{attribute 'linkalways'} 
{attribute 'no_explicit_call' := 'This FB is a CLASS and must be accessed using methods or properties'}
{attribute 'enable_dynamic_creation'}
FUNCTION_BLOCK _ETcVnFontType EXTENDS EnumDatatypeBase
VAR
	localData : ETcVnFontType;
	activeData : REFERENCE TO ETcVnFontType;
	enumBaseDatatype : _DINT(localData);
END_VAR

METHOD PRIVATE AddLocalEnumeration
VAR_INPUT
	Enumeration : T_MAXSTRING;
	Value : ETcVnFontType;
END_VAR
AddEnumeration(Enumeration, Value);
END_METHOD

PROPERTY PUBLIC Address : PVOID
GET
Address := ADR(activeData);
END_GET
END_PROPERTY

METHOD PUBLIC ClearReference
VAR_INPUT
END_VAR
activeData REF= localData;
SetBaseDatatypeReference();
END_METHOD

METHOD PUBLIC Clone : I_Datatype
VAR
    pClone : POINTER TO _ETcVnFontType;
END_VAR
pClone := __NEW(_ETcVnFontType(InitialValue := Value));
Clone := pClone^;
END_METHOD

METHOD FB_init : BOOL
VAR_INPUT
	bInitRetains : BOOL; // if TRUE, the retain variables are initialized (warm start / cold start)
	bInCopyCode : BOOL;  // if TRUE, the instance afterwards gets moved into the copy code (online change)
	InitialValue : ETcVnFontType;
END_VAR
localData := InitialValue;
AddBaseDatatype(enumBaseDatatype);
ClearReference();

AddLocalEnumeration('TCVN_FT_HERSHEY_SIMPLEX', ETcVnFontType.TCVN_FT_HERSHEY_SIMPLEX);
AddLocalEnumeration('TCVN_FT_HERSHEY_PLAIN', ETcVnFontType.TCVN_FT_HERSHEY_PLAIN);
AddLocalEnumeration('TCVN_FT_HERSHEY_DUPLEX', ETcVnFontType.TCVN_FT_HERSHEY_DUPLEX);
AddLocalEnumeration('TCVN_FT_HERSHEY_COMPLEX', ETcVnFontType.TCVN_FT_HERSHEY_COMPLEX);
AddLocalEnumeration('TCVN_FT_HERSHEY_TRIPLEX', ETcVnFontType.TCVN_FT_HERSHEY_TRIPLEX);
AddLocalEnumeration('TCVN_FT_HERSHEY_COMPLEX_SMALL', ETcVnFontType.TCVN_FT_HERSHEY_COMPLEX_SMALL);
AddLocalEnumeration('TCVN_FT_HERSHEY_SCRIPT_SIMPLEX', ETcVnFontType.TCVN_FT_HERSHEY_SCRIPT_SIMPLEX);
AddLocalEnumeration('TCVN_FT_HERSHEY_SCRIPT_COMPLEX', ETcVnFontType.TCVN_FT_HERSHEY_SCRIPT_COMPLEX);
AddLocalEnumeration('TCVN_FT_HERSHEY_PLAIN_ITALIC', ETcVnFontType.TCVN_FT_HERSHEY_PLAIN_ITALIC);
AddLocalEnumeration('TCVN_FT_HERSHEY_COMPLEX_ITALIC', ETcVnFontType.TCVN_FT_HERSHEY_COMPLEX_ITALIC);
AddLocalEnumeration('TCVN_FT_HERSHEY_TRIPLEX_ITALIC', ETcVnFontType.TCVN_FT_HERSHEY_TRIPLEX_ITALIC);
AddLocalEnumeration('TCVN_FT_HERSHEY_COMPLEX_SMALL_ITALIC', ETcVnFontType.TCVN_FT_HERSHEY_COMPLEX_SMALL_ITALIC);
END_METHOD

PROPERTY PUBLIC Identifier : T_MAXSTRING
GET
Identifier := 'ETcVnFontType';
END_GET
END_PROPERTY

METHOD IsEnumeratorValueEqual : BOOL
VAR_INPUT
	Enumerator : I_KeyValueForwardEnumerator;
END_VAR
VAR
	storedValue : ETcVnFontType;
END_VAR
IF NOT Enumerator.TryGet(storedValue) THEN
	RETURN;
END_IF

IsEnumeratorValueEqual := storedValue = activeData;
END_METHOD

METHOD PUBLIC MakeReferenceTo
VAR_INPUT
	ReferenceTarget : REFERENCE TO ETcVnFontType;
END_VAR
activeData REF= ReferenceTarget;
SetBaseDatatypeReference();
END_METHOD

METHOD PROTECTED SetBaseDatatypeReference
VAR_INPUT
END_VAR
enumBaseDatatype.MakeReferenceTo(activeData);
END_METHOD

PROPERTY PUBLIC Size : UDINT
GET
Size := SIZEOF(activeData);
END_GET
END_PROPERTY

METHOD TryMakeReferenceTo : BOOL
VAR_INPUT
	Target : I_Datatype;
END_VAR
VAR
	targetAsEnum : I_EnumDatatype;
	pTargetData : POINTER TO ETcVnFontType;
END_VAR
IF NOT Target.TryResolveAsEnumDatatype(targetAsEnum) THEN
	RETURN;
END_IF

IF targetAsEnum.Identifier <> Identifier THEN
	RETURN;
END_IF

pTargetData := Target.Address;
activeData REF= pTargetData^;
SetBaseDatatypeReference();
TryMakeReferenceTo := TRUE;
END_METHOD

PROPERTY PUBLIC Value : ETcVnFontType
GET
Value := activeData;
END_GET
SET
activeData := Value;
END_SET
END_PROPERTY

END_FUNCTION_BLOCK

(* stored: Version 1.1.0.1, ProductVersion 3.1.4024.12
   POU _ETcVnFontType: Id {3d30620a-6fbf-49c2-aa5e-f1c2d9427120}, SpecialFunc None
   Folder Constructor: Id {ee00bf30-bb95-4ab6-93b9-dc7a7a5bad36}
   Folder Private: Id {c5e8bc94-e735-4db7-9d22-0e72df6e2c7a}
   Folder Protected: Id {c74f9896-74e4-42b4-aad7-25349e49f7b2}
   Method AddLocalEnumeration: Id {dd478bdd-f1c9-4660-9c66-8731fc071532}
   Property Address: Id {d814ecd6-78b8-4405-9a5b-34e36eb75189}
   Get Get: Id {50b03b9c-064e-48aa-b6d2-c7bfdd664038}
   Method ClearReference: Id {8aca728f-60dd-44d2-bf04-96ef497d1692}
   Method Clone: Id {79de8ef4-bd0e-4445-972e-9c11bbaacafb}
   Method FB_init: Id {6860cb2b-a0c5-4ee9-9787-f99d0a1d5756}
   Property Identifier: Id {173e90d3-c0cd-48c0-a46d-dbb29fc9af6e}
   Get Get: Id {62d7d615-4b59-4df4-8aba-43579a5296cf}
   Method IsEnumeratorValueEqual: Id {1ed78b49-4386-4375-9a05-1c4bf971aa7b}
   Method MakeReferenceTo: Id {196fd061-b9a1-4952-9097-9517d0abfc65}
   Method SetBaseDatatypeReference: Id {ee2766cd-bfa2-49cc-bf40-09edd9e6b362}
   Property Size: Id {3fb96b77-e494-4516-b7c0-f5306ae69574}
   Get Get: Id {96becf50-df54-43e7-8f46-dfbac5bf0e7c}
   Method TryMakeReferenceTo: Id {99ef0f53-425c-42c7-b275-cb2b8f366efc}
   Property Value: Id {36451213-0006-4f54-829f-8d4d6ca65bcc}
   Get Get: Id {93311820-7953-492a-a46f-3860be3eba42}
   Set Set: Id {e802dd1a-96d4-41d5-a7f2-ef63af0e2b89} *)
